FUNCTION_BLOCK FB_Event IMPLEMENTS I_Event
VAR_INPUT
	fbObserver:			FB_Observable;				// Observer
END_VAR
VAR_OUTPUT
END_VAR
VAR
	{IF (defined (release))}
    	{attribute 'hide'}
	{END_IF}
	iLogger:			I_Logger;					// Event logger
	{IF (defined (release))}
    	{attribute 'hide'}
	{END_IF}
	iParent:			I_Element;					// Parent component
	{IF (defined (release))}
    	{attribute 'hide'}
	{END_IF}
	fbList:				FB_ListString;				// contains a list with string values
	stDebug:			ST_Event;					// last debug event
	stInfo:				ST_Event;					// last info event
	stWarning:			ST_Event;					// last warning event
	stError:			ST_Event;					// last error event
	stFatal:			ST_Event;					// last Fatal event
END_VAR

// https://peterzerlauth.com/
fbObserver();

METHOD FB_init : BOOL
VAR_INPUT
	bInitRetains : BOOL; // if TRUE, the retain variables are initialized (warm start / cold start)
	bInCopyCode : BOOL;  // if TRUE, the instance afterwards gets moved into the copy code (online change)
	iParent:			I_Element;
END_VAR
THIS^.iParent:= iParent;
fbObserver.iParent:= iParent;
END_METHOD

METHOD PUBLIC M_AddBOOL : I_Event
VAR_INPUT
	Value: 	bool;
END_VAR
fbList.M_Add(BOOL_TO_STRING(Value));
M_AddBOOL:= THIS^;
END_METHOD

METHOD PUBLIC M_AddINT : I_Event
VAR_INPUT
	Value: 	LINT;
END_VAR
fbList.M_Add(LINT_TO_STRING(Value));
M_AddINT:= THIS^;
END_METHOD

METHOD PUBLIC M_AddREAL : I_Event
VAR_INPUT
	Value: 	Lreal;
	Decimals: INT;
END_VAR
fbList.M_Add(LREAL_TO_FMTSTR(Value, Decimals, TRUE));
M_AddREAL:= THIS^;
END_METHOD

METHOD PUBLIC M_AddSTRING : I_Event
VAR_INPUT
	Value: STRING(255);
END_VAR
fbList.M_Add(Value);
M_AddSTRING:= THIS^;
END_METHOD

METHOD PUBLIC M_AddTIME : I_Event
VAR_INPUT
	Value: 	TIME;
END_VAR
fbList.M_Add(TIME_TO_STRING(Value));
M_AddTIME:= THIS^;
END_METHOD

METHOD INTERNAL M_Arguments : STRING(255)
VAR_INPUT
END_VAR
VAR
	nIndex:			INT;
END_VAR
WHILE nIndex < fbList. P_Length DO
	M_Arguments:= Concat(Concat(M_Arguments, fbList.M_Index(nIndex)), '$N');
	nIndex:= nIndex + 1;
END_WHILE

fbList.M_Clear();
END_METHOD

METHOD INTERNAL M_Build : STRING(255)
VAR_INPUT
	sMessage:		STRING(255);
END_VAR
VAR
	nIndex:		   	DINT;
	nPosition: 		INT;
END_VAR
nPosition:= Find(sMessage, '%s');
WHILE nPosition <> 0 DO
	sMessage:= Replace(sMessage, fbList.M_Index(nIndex), 2, nPosition);
	nPosition:= Find(sMessage, '%s');
	nIndex:= nIndex + 1;
END_WHILE
M_Build:= sMessage;
END_METHOD

METHOD PUBLIC M_Debug
VAR_INPUT
	sMessage:				STRING(255);
END_VAR
stDebug.sMessage:= sMessage;
stDebug.iSource:= iParent;
stDebug.sInstance:= iParent.P_Reflection.P_Instance;
stDebug.sClass:= iParent.P_Reflection.P_Class;
stDebug.eEventType:= E_Event.Debug;
stDebug.tTimestamp:= iParent.P_Reflection.P_Timestamp;
stDebug.nID:= 0;
stDebug.sDefault:= M_Build(sMessage);
stDebug.sArguments:= M_Arguments();
stDebug.stFlags.bActive:= TRUE;
stDebug.stFlags.bRemove:= TRUE;

IF iLogger = 0 THEN
	M_Log(stDebug);
ELSE
	iLogger.M_Log(stDebug);
END_IF
END_METHOD

METHOD PUBLIC M_Error
VAR_INPUT
	sMessage:				STRING(255);
	nID:					ULINT;
END_VAR
stError.sMessage:= sMessage;
stError.iSource:= iParent;
stError.sInstance:= iParent.P_Reflection.P_Instance;
stError.sClass:= iParent.P_Reflection.P_Class;
stError.eEventType:= E_Event.Error;
stError.tTimestamp:= iParent.P_Reflection.P_Timestamp;
stError.nID:= nID;
stError.sDefault:= M_Build(sMessage);
stError.sArguments:= M_Arguments();
stError.stFlags.bActive:= TRUE;
stError.stFlags.bRemove:= FALSE;

IF iLogger = 0 THEN
	M_Log(stError);
ELSE
	iLogger.M_Log(stError);
END_IF
END_METHOD

METHOD PUBLIC M_Fatal
VAR_INPUT
	sMessage:				STRING(255);
	nID:					ULINT;
END_VAR
stFatal.sMessage:= sMessage;
stFatal.iSource:= iParent;
stFatal.sInstance:= iParent.P_Reflection.P_Instance;
stFatal.sClass:= iParent.P_Reflection.P_Class;
stFatal.eEventType:= E_Event.Error;
stFatal.tTimestamp:= iParent.P_Reflection.P_Timestamp;
stFatal.nID:= nID;
stFatal.sDefault:= M_Build(sMessage);
stFatal.sArguments:= M_Arguments();
stFatal.stFlags.bActive:= TRUE;
stFatal.stFlags.bRemove:= FALSE;

IF iLogger = 0 THEN
	M_Log(stFatal);
ELSE
	iLogger.M_Log(stFatal);
END_IF

fbObserver.M_Notify(iParent);
END_METHOD

METHOD PUBLIC M_Info
VAR_INPUT
	sMessage:				STRING(255);
	nID:					ULINT;
END_VAR
stInfo.sMessage:= sMessage;
stInfo.iSource:= iParent;
stInfo.sInstance:= iParent.P_Reflection.P_Instance;
stInfo.sClass:= iParent.P_Reflection.P_Class;
stInfo.eEventType:= E_Event.Information;
stInfo.tTimestamp:= iParent.P_Reflection.P_Timestamp;
stInfo.nID:= nID;
stInfo.sDefault:= M_Build(sMessage);
stInfo.sArguments:= M_Arguments();
stInfo.stFlags.bActive:= TRUE;
stInfo.stFlags.bRemove:= TRUE;

IF iLogger = 0 THEN
	M_Log(stInfo);
ELSE
	iLogger.M_Log(stInfo);
END_IF
END_METHOD

METHOD PRIVATE M_Log : BOOL
VAR_INPUT
	stEvent	: ST_Event;
END_VAR
END_METHOD

METHOD PUBLIC M_Warning
VAR_INPUT
	sMessage:				STRING(255);
	nID:					ULINT;
END_VAR
stWarning.sMessage:= sMessage;
stWarning.iSource:= iParent;
stWarning.sInstance:= iParent.P_Reflection.P_Instance;
stWarning.sClass:= iParent.P_Reflection.P_Class;
stWarning.eEventType:= E_Event.Warning;
stWarning.tTimestamp:= iParent.P_Reflection.P_Timestamp;
stWarning.nID:= nID;
stWarning.sDefault:= M_Build(sMessage);
stWarning.sArguments:= M_Arguments();
stWarning.stFlags.bActive:= TRUE;
stWarning.stFlags.bRemove:= TRUE;

IF iLogger = 0 THEN
	M_Log(stWarning);
ELSE
	iLogger.M_Log(stWarning);
END_IF
END_METHOD

{attribute 'OPC.UA.DA.Property' := '1'}
{attribute 'monitoring' := 'call'}
PROPERTY P_Logger : I_Logger
GET
P_Logger:= iLogger;
END_GET
SET
iLogger:= P_Logger;
END_SET
END_PROPERTY

{attribute 'OPC.UA.DA.Property' := '1'}
{attribute 'monitoring' := 'call'}
PROPERTY PUBLIC P_Observer : I_Observable
GET
P_Observer:= fbObserver;
END_GET
END_PROPERTY

END_FUNCTION_BLOCK

(* stored: Version 1.1.0.1
   POU FB_Event: Id {59616103-7f2e-4b6f-81bd-583969a36d28}, SpecialFunc None
   Method FB_init: Id {be23ffcc-529d-4010-ace3-b17baed191a5}
   Method M_AddBOOL: Id {55367f5b-ac71-0a63-095c-881721842948}
   Method M_AddINT: Id {77c01fd5-65e9-07ed-2cff-a79b9d444c15}
   Method M_AddREAL: Id {b0c25678-4933-0839-34f0-c4eb0def69fb}
   Method M_AddSTRING: Id {8ae81d27-cb47-01bb-2b19-fe8608e777a8}
   Method M_AddTIME: Id {a7c2a656-d860-0eb9-0cff-1e8b5b1d8573}
   Method M_Arguments: Id {70779266-7b36-4bce-9e6f-049e951fd75a}
   Method M_Build: Id {c94cd0c6-56df-0b94-2d8d-b10a55caeb26}
   Method M_Debug: Id {0a2b992b-2a4a-0251-0210-713b326debf6}
   Method M_Error: Id {20d0062d-a518-02ec-13ef-e4c8c4295653}
   Method M_Fatal: Id {a968dc5e-d8ee-079a-0799-c81d1c9d2558}
   Method M_Info: Id {d9a244f2-1d6f-434f-aab4-cad6aacbb94f}
   Method M_Log: Id {4faf2127-0b92-014c-3fdc-3aa74f15a00e}
   Method M_Warning: Id {d443b8bb-774e-487e-80a2-79cf66a0376c}
   Property P_Logger: Id {7db5ebbd-2df4-0da4-1172-1f7f59531c54}
   Get Get: Id {c30909c8-bc71-0c3f-2d6b-a056f1f6fe1b}
   Set Set: Id {69321800-5ac3-0207-1f07-4cc88412ab84}
   Property P_Observer: Id {5a2ea21c-aedb-0c6a-2f12-df08356b98aa}
   Get Get: Id {a355a491-866b-0089-1d02-e50cef149847} *)
